FUNCTION_BLOCK FB_Blinker
VAR_INPUT

	bStart									:BOOL;
	tTurnOnDelay							:TIME;
	tTurnOffDelay							:TIME;

END_VAR
VAR_OUTPUT

	bLed									:BOOL;

END_VAR
VAR

	fbTimer1								:TON;
	fbTimer2								:TON;

END_VAR
(* End *)

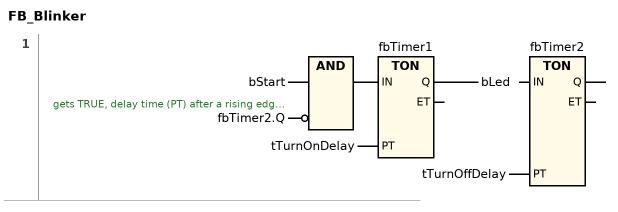
// NETWORK 1
//   fbTimer2.Q: gets TRUE, delay time (PT) after a rising edge at IN
fbTimer1(IN := bStart AND NOT fbTimer2.Q, PT := tTurnOnDelay); // TON
bLed := fbTimer1.Q;
fbTimer2(IN := fbTimer1.Q, PT := tTurnOffDelay); // TON

END_FUNCTION_BLOCK

(* stored: Version 1.1.0.1
   POU FB_Blinker: Id {f88f028e-0da1-49a3-90fb-a7fb86d3d0fd}, SpecialFunc None *)
